// TIA Portal project "TrattamentiTermici" (V18)

(* hardware
DEVICE "S71500/ET200MP station_1"  S7-1500 station
   slot 0: "Telaio di montaggio_0"  Rack  6ES7 590-1***0-0AA0
   slot 1: "PLC_1"  CPU 1516-3 PN/DP  6ES7 516-3AN01-0AB0  V2.5
      slot 3: "Display CPU_1"  6ES7591-1BA00-0AA0
   slot 2: "DI 32x24VDC HF_1"  DI 32x24VDC HF  6ES7 521-1BL00-0AB0  V2.1
   slot 3: "DQ 32x24VDC/0.5A HF_1"  DQ 32x24VDC/0.5A HF  6ES7 522-1BL01-0AB0  V1.0
   slot 4: "AI 8xU/I/RTD/TC ST_1"  AI 8xU/I/RTD/TC ST  6ES7 531-7KF00-0AB0  V2.1
   slot 5: "AQ 4xU/I ST_1"  AQ 4xU/I ST  6ES7 532-5HD00-0AB0  V2.1
*)

// ===== PLC "PLC_1"  CPU 1516-3 PN/DP =====

VAR_GLOBAL   // PLC tag table "Tabella delle variabili standard"
   "AperturaCoperchio" AT %Q0.0 : Bool;
   "ChiusuraCoperchio" AT %Q0.1 : Bool;
   "DiscesaPunta" AT %Q0.2 : Bool;
   "AbbassaBraccio" AT %Q0.3 : Bool;
   "LedEmergenza" AT %Q0.4 : Bool;
   "MotoreIndietro" AT %Q0.5 : Bool;
   "MotoreAvanti" AT %Q0.6 : Bool;
   "SalitaPunta" AT %Q0.7 : Bool;
   "AlzaBraccio" AT %Q1.0 : Bool;
   "led11" AT %Q1.1 : Bool;
   "led12" AT %Q1.2 : Bool;
   "led13" AT %Q1.3 : Bool;
   "led14" AT %Q1.4 : Bool;
   "led15" AT %Q1.5 : Bool;
   "led16" AT %Q1.6 : Bool;
   "led17" AT %Q1.7 : Bool;
   "led20" AT %Q2.0 : Bool;
   "led21" AT %Q2.1 : Bool;
   "led22" AT %Q2.2 : Bool;
   "led23" AT %Q2.3 : Bool;
   "led24" AT %Q2.4 : Bool;
   "led25" AT %Q2.5 : Bool;
   "led26" AT %Q2.6 : Bool;
   "led27" AT %Q2.7 : Bool;
   "led30" AT %Q3.0 : Bool;
   "led31" AT %Q3.1 : Bool;
   "led32" AT %Q3.2 : Bool;
   "led33" AT %Q3.3 : Bool;
   "led34" AT %Q3.4 : Bool;
   "led35" AT %Q3.5 : Bool;
   "led36" AT %Q3.6 : Bool;
   "led37" AT %Q3.7 : Bool;
   "BraccioSu" AT %I0.2 : Bool;
   "BraccioGiu" AT %I0.3 : Bool;
   "FotocellulaSinistra" AT %I0.4 : Bool;
   "FotocellulaCentrale" AT %I0.5 : Bool;
   "FotocellulaDestra" AT %I0.6 : Bool;
   "PulsanteInizializzazione" AT %I0.7 : Bool;
   "PulsanteMarcia" AT %I1.0 : Bool;
   "PulsanteStop" AT %I1.1 : Bool;
   "PulsanteEmergenza" AT %I1.2 : Bool;
   "CoperchioAperto" AT %I2.1 : Bool;
END_VAR

DATA_BLOCK "DB_Comandi"   // DB1
{ S7_Optimized_Access := 'FALSE' }
VERSION : 0.1
   VAR
      bStop : Bool;
      bAuto : Bool;
      bMan : Bool;
      bReset : Bool;
      bEmergenza : Bool;
   END_VAR
BEGIN
END_DATA_BLOCK

DATA_BLOCK "DB_Stati"   // DB2
{ S7_Optimized_Access := 'FALSE' }
VERSION : 0.1
   VAR
      sAuto : Bool;
      sStop : Bool;
      sMan : Bool;
      sHome : Bool;
      sAttesastop : Bool;
      sEmergenza : Bool;
      bIni1 : Bool;
      bIni2 : Bool;
      bRip1 : Bool;
      bRip2 : Bool;
   END_VAR
BEGIN
END_DATA_BLOCK

DATA_BLOCK "DB_Tappe"   // DB3
{ S7_Optimized_Access := 'FALSE' }
VERSION : 0.1
   VAR
      tappeGemma : Int;
      tappeM1 : Int;
   END_VAR
BEGIN
END_DATA_BLOCK

DATA_BLOCK "DB_Variabili"   // DB4
{ S7_Optimized_Access := 'FALSE' }
VERSION : 0.1
   VAR
      timerResetPulsantiSTART : Bool;
      timerResetPulsantiDONE : Bool;
      timerResetPulsantiOUTPUT : Time;
      timerResetPulsantiDURATA : Time;
      BraccioSu : Bool;
      BraccioGiu : Bool;
      FotocellulaSinistra : Bool;
      FotocellulaCentrale : Bool;
      FotocellulaDestra : Bool;
      BtnInizio : Bool;
      BtnMarcia : Bool;
      BtnStop : Bool;
      BtnEmergenza : Bool;
      CoperchioAperto : Bool;
      AperturaCoperchio : Bool;
      ChiusuraCoperchio : Bool;
      DiscesaPunta : Bool;
      AbbassaBraccio : Bool;
      LedEmergenza : Bool;
      MotoreIndietro : Bool;
      MotoreAvanti : Bool;
      AlzaBraccio : Bool;
      SalitaPunta : Bool;
      nShake : Int;
      nPezzi : Int;
      giaAumentato : Bool;
   END_VAR
BEGIN
END_DATA_BLOCK

// folder: System blocks/Program resources

DATA_BLOCK "timerResetPulsanti"   // DB5
{ S7_Optimized_Access := 'TRUE' }
AUTHOR : Simatic
FAMILY : IEC
NAME : IEC_TMR
VERSION : 1.0
// stored: InstanceOfName IEC_TIMER
"IEC_TIMER"
BEGIN
END_DATA_BLOCK

// folder: (top level)

FUNCTION "FC_Gemma" : Void   // FC1, SCL
{ S7_Optimized_Access := 'TRUE' }
VERSION : 0.1
BEGIN
   CASE "DB_Tappe".tappeGemma OF
       0:  //Stato di riposo
           "DB_Stati".sStop := TRUE;
           IF "DB_Comandi".bAuto = TRUE THEN
               "DB_Tappe".tappeGemma := 1;//home
               "DB_Stati".sAuto := FALSE;
               "DB_Stati".sHome := TRUE;
               "DB_Stati".sMan := FALSE;
               "DB_Stati".sStop := FALSE;
               "DB_Stati".sEmergenza := FALSE;
           ELSE
               IF "DB_Comandi".bMan = TRUE THEN
                   "DB_Tappe".tappeGemma := 4;//home
                   "DB_Stati".sAuto := FALSE;
                   "DB_Stati".sHome := FALSE;
                   "DB_Stati".sMan := TRUE;
                   "DB_Stati".sStop := FALSE;
                   "DB_Stati".sEmergenza := FALSE;
               END_IF;
           END_IF;
          1: //Stato di home
              IF "DB_Stati".bIni1 = TRUE AND "DB_Stati".bIni2 = TRUE THEN
                  "DB_Tappe".tappeGemma := 2;//automatico
                  "DB_Stati".sAttesastop := TRUE;
                  "DB_Stati".sAuto := TRUE;
                  "DB_Stati".sHome := FALSE;
                  "DB_Stati".sMan := FALSE;
                  "DB_Stati".sStop := FALSE;
                  "DB_Stati".sEmergenza := FALSE;
              END_IF;
          2: //Stato di automatico
              IF "DB_Comandi".bStop = TRUE THEN
                  "DB_Tappe".tappeGemma := 3;//attesa stop
                  "DB_Stati".sAttesastop := TRUE;
                  "DB_Stati".sAuto := FALSE;
                  "DB_Stati".sHome := FALSE;
                  "DB_Stati".sMan := FALSE;
                  "DB_Stati".sStop := FALSE;
                  "DB_Stati".sEmergenza := FALSE;
              END_IF;
          3: //Stato di attesa stop
              IF "DB_Stati".bRip1 = TRUE AND "DB_Stati".bRip2 = TRUE THEN
                  "DB_Tappe".tappeGemma := 0;//stop
                  "DB_Stati".sAttesastop := TRUE;
                  "DB_Stati".sAuto := FALSE;
                  "DB_Stati".sHome := FALSE;
                  "DB_Stati".sMan := FALSE;
                  "DB_Stati".sStop := TRUE;
                  "DB_Stati".sEmergenza := FALSE;
              END_IF;
          4: //Stato di manuale
              IF "DB_Comandi".bStop = TRUE = TRUE THEN
                  "DB_Tappe".tappeGemma := 0;//stop
                  "DB_Stati".sAuto := FALSE;
                  "DB_Stati".sHome := FALSE;
                  "DB_Stati".sMan := FALSE;
                  "DB_Stati".sStop := TRUE;
                  "DB_Stati".sEmergenza := FALSE;
              END_IF;
          5: //Stato di emergenza
              IF "DB_Comandi".bEmergenza = TRUE AND "DB_Stati".sEmergenza = TRUE THEN
                  "DB_Tappe".tappeGemma := 0;//stop
                  "DB_Stati".sAuto := FALSE;
                  "DB_Stati".sHome := FALSE;
                  "DB_Stati".sMan := FALSE;
                  "DB_Stati".sStop := TRUE;
                  "DB_Stati".sEmergenza := FALSE;
              END_IF;
      END_CASE;
   //gestione emergenza

      IF "DB_Comandi".bEmergenza = FALSE THEN
          "DB_Tappe".tappeGemma := 5;//emergenza
      "DB_Stati".sAttesastop := FALSE;
      "DB_Stati".sAuto := FALSE;
      "DB_Stati".sHome := FALSE;
      "DB_Stati".sMan := FALSE;
      "DB_Stati".sStop := FALSE;
      "DB_Stati".sEmergenza := TRUE;
   END_IF;
END_FUNCTION

FUNCTION "FC_Grafcet" : Void   // FC2, SCL
{ S7_Optimized_Access := 'TRUE' }
VERSION : 0.1
BEGIN
   //Imposto bRini e bRip a TRUE. Andranno poi gestiti in base alle condizioni dell'impianto
   "DB_Stati".bIni1 := TRUE;
   "DB_Stati".bIni2 := TRUE;
   "DB_Stati".bRip1 := TRUE;
   "DB_Stati".bRip2 := TRUE;
   //
   //gestico il RESET
   //

   IF "DB_Tappe".tappeM1 = 0 THEN
       IF "DB_Stati".sAuto AND "DB_Stati".bIni1 AND "DB_Stati".sAttesastop THEN
           "DB_Tappe".tappeM1 := 1;
       END_IF;

       "DB_Variabili".nPezzi := 0;
       "DB_Variabili".timerResetPulsantiDURATA := T#400ms;
   END_IF;

   IF "DB_Tappe".tappeM1 = 1 THEN
       "DB_Variabili".AlzaBraccio := TRUE;

       IF "DB_Variabili".BraccioSu  THEN
           "DB_Variabili".AlzaBraccio := FALSE;
           "DB_Variabili".MotoreAvanti := TRUE;
       END_IF;

       IF "DB_Variabili".FotocellulaCentrale=TRUE THEN
           "DB_Variabili".MotoreAvanti := FALSE;
           "DB_Tappe".tappeM1 := 2;
       END_IF;
   END_IF;

   IF "DB_Tappe".tappeM1 = 2 THEN
       "DB_Variabili".AbbassaBraccio := TRUE;
       "DB_Variabili".nShake := 0;

       IF "DB_Variabili".BraccioGiu THEN
           "DB_Variabili".AbbassaBraccio := FALSE;
           "DB_Tappe".tappeM1 := 3;
           "DB_Variabili".nShake := 0;
       END_IF;
   END_IF;


   IF "DB_Tappe".tappeM1 = 3 THEN
       "DB_Variabili".DiscesaPunta := TRUE;
       "DB_Variabili".timerResetPulsantiDURATA := T#400ms;
       "DB_Variabili".timerResetPulsantiSTART := TRUE;

       IF "DB_Variabili".timerResetPulsantiDONE THEN
           "DB_Variabili".timerResetPulsantiSTART := FALSE;
           "DB_Variabili".timerResetPulsantiDONE := FALSE;
           "DB_Variabili".giaAumentato := FALSE;
           "DB_Variabili".DiscesaPunta := FALSE;
           "DB_Tappe".tappeM1 := 4;
       END_IF;
   END_IF;

   IF "DB_Tappe".tappeM1 = 4 THEN
       "DB_Variabili".SalitaPunta := TRUE;
       "DB_Variabili".timerResetPulsantiSTART := TRUE;
       "DB_Variabili".timerResetPulsantiDURATA := T#400ms;

       IF "DB_Variabili".timerResetPulsantiDONE THEN
           IF "DB_Variabili".giaAumentato=FALSE THEN
               "DB_Variabili".nShake += 1;
               "DB_Variabili".giaAumentato := TRUE;
               "DB_Variabili".SalitaPunta := FALSE;
           END_IF;
           IF "DB_Variabili".nShake = 6 THEN
               "DB_Variabili".AlzaBraccio := TRUE;
               IF "DB_Variabili".BraccioSu THEN
                   "DB_Variabili".AlzaBraccio := FALSE;
                   "DB_Variabili".timerResetPulsantiSTART := FALSE;
                   "DB_Variabili".timerResetPulsantiDONE := FALSE;
                   "DB_Tappe".tappeM1 := 5;
               END_IF;
           ELSE
               "DB_Tappe".tappeM1 := 3;
           END_IF;
       END_IF;
   END_IF;

   IF "DB_Tappe".tappeM1 = 5 THEN
       "DB_Variabili".AperturaCoperchio := TRUE;
       "DB_Variabili".MotoreAvanti := TRUE;

       IF "DB_Variabili".FotocellulaDestra = TRUE THEN
           "DB_Variabili".AperturaCoperchio := FALSE;
           "DB_Variabili".MotoreAvanti := FALSE;
           "DB_Tappe".tappeM1 := 6;
       END_IF;
   END_IF;

   IF "DB_Tappe".tappeM1 = 6 THEN
       "DB_Variabili".AbbassaBraccio := TRUE;

       IF "DB_Variabili".BraccioGiu THEN
           "DB_Variabili".AbbassaBraccio := FALSE;
           "DB_Variabili".DiscesaPunta := TRUE;
           "DB_Variabili".timerResetPulsantiSTART := TRUE;
           "DB_Variabili".timerResetPulsantiDURATA := T#3000ms;
       END_IF;

       IF "DB_Variabili".timerResetPulsantiDONE THEN
           "DB_Variabili".DiscesaPunta := FALSE;
           "DB_Variabili".timerResetPulsantiSTART := FALSE;
           "DB_Variabili".timerResetPulsantiDONE := FALSE;
           "DB_Tappe".tappeM1 := 7;
       END_IF;
   END_IF;

   IF "DB_Tappe".tappeM1 = 7 THEN
       "DB_Variabili".SalitaPunta := TRUE;
       "DB_Variabili".AlzaBraccio := TRUE;

       IF "DB_Variabili".BraccioSu THEN
           "DB_Variabili".SalitaPunta := FALSE;
           "DB_Variabili".AlzaBraccio := FALSE;
           "DB_Tappe".tappeM1 := 8;
           "DB_Variabili".nPezzi+=1;
       END_IF;
       ;
   END_IF;

   IF "DB_Tappe".tappeM1 = 8 THEN
       "DB_Variabili".MotoreIndietro := TRUE;

       IF "DB_Variabili".FotocellulaCentrale THEN
           "DB_Variabili".MotoreIndietro := FALSE;
           "DB_Tappe".tappeM1 := 9;
       END_IF;
       ;
   END_IF;

   IF "DB_Tappe".tappeM1 = 9 THEN
       "DB_Variabili".MotoreIndietro := TRUE;
       "DB_Variabili".ChiusuraCoperchio := TRUE;

       IF "DB_Variabili".FotocellulaSinistra THEN
           "DB_Variabili".MotoreIndietro := FALSE;
           "DB_Variabili".timerResetPulsantiSTART := TRUE;
           "DB_Variabili".timerResetPulsantiDONE := FALSE;
           "DB_Variabili".timerResetPulsantiDURATA := T#5000ms;
       END_IF;

       IF "DB_Variabili".timerResetPulsantiDONE THEN
           "DB_Variabili".timerResetPulsantiSTART := FALSE;
           "DB_Variabili".timerResetPulsantiDONE := FALSE;
           "DB_Tappe".tappeM1 := 0;
           "DB_Variabili".ChiusuraCoperchio := FALSE;
       END_IF;
   END_IF;
END_FUNCTION

FUNCTION "FC_ResetPulsanti" : Void   // FC3, SCL
{ S7_Optimized_Access := 'TRUE' }
VERSION : 0.1
BEGIN
   IF "DB_Comandi".bAuto = TRUE OR
       "DB_Comandi".bMan = TRUE OR
       "DB_Comandi".bReset = TRUE OR
       "DB_Comandi".bStop = TRUE THEN
       //
       "DB_Variabili".timerResetPulsantiSTART := TRUE;
   END_IF;
   IF "DB_Variabili".timerResetPulsantiDONE = TRUE THEN
       "DB_Variabili".timerResetPulsantiSTART := FALSE;
       "DB_Variabili".timerResetPulsantiDONE := FALSE;
       "DB_Comandi".bAuto := FALSE;
       "DB_Comandi".bMan := FALSE;
       "DB_Comandi".bReset := FALSE;
       "DB_Comandi".bStop := FALSE;
   END_IF;
END_FUNCTION

FUNCTION "FC_Timer" : Void   // FC4, SCL
{ S7_Optimized_Access := 'TRUE' }
VERSION : 0.1
BEGIN
   "DB_Variabili".timerResetPulsantiDURATA := T#400ms;
   "timerResetPulsanti".TON(IN:="DB_Variabili".timerResetPulsantiSTART,
                            PT:="DB_Variabili".timerResetPulsantiDURATA,
                            Q=>"DB_Variabili".timerResetPulsantiDONE,
                            ET=>"DB_Variabili".timerResetPulsantiOUTPUT);
END_FUNCTION

FUNCTION "FC_Uscite" : Void   // FC5, SCL
{ S7_Optimized_Access := 'TRUE' }
VERSION : 0.1
BEGIN
   //prima di scrivere fisicamente le uscite
   //devo controllare che tutte le condizioni
   //siano rispettate
   //emergenza, protezioni, fotocellule ecc.
   "AperturaCoperchio" := "DB_Variabili".ChiusuraCoperchio;
   "ChiusuraCoperchio" := "DB_Variabili".AperturaCoperchio;
   "DiscesaPunta" := "DB_Variabili".AbbassaBraccio;
   "AbbassaBraccio" := "DB_Variabili".DiscesaPunta;
   "LedEmergenza" := "DB_Variabili".LedEmergenza;
   "MotoreIndietro" := "DB_Variabili".MotoreIndietro;
   "MotoreAvanti" := "DB_Variabili".MotoreAvanti;
   "AlzaBraccio" := "DB_Variabili".AlzaBraccio;
   "SalitaPunta" := "DB_Variabili".SalitaPunta;

   // Uscite
   "DB_Variabili".BraccioSu := "BraccioSu";
   "DB_Variabili".BraccioGiu := "BraccioGiu";
   "DB_Variabili".FotocellulaSinistra := "FotocellulaSinistra";
   "DB_Variabili".FotocellulaCentrale := "FotocellulaCentrale";
   "DB_Variabili".FotocellulaDestra := "FotocellulaDestra";
   "DB_Variabili".BtnInizio := "PulsanteMarcia";
   "DB_Variabili".BtnStop := "PulsanteStop";
   "DB_Variabili".BtnEmergenza := "PulsanteEmergenza";
   "DB_Variabili".CoperchioAperto :="CoperchioAperto";
END_FUNCTION

ORGANIZATION_BLOCK "Main"   // OB1, LAD, ProgramCycle
TITLE = "Main Program Sweep (Cycle)"
{ S7_Optimized_Access := 'TRUE' }
VERSION : 0.1
   VAR_INPUT
      Initial_Call : Bool;   // Initial call of this OB
      Remanence : Bool;   // =True, if remanent data are available
   END_VAR
   VAR_TEMP   // added for the SCL form of the ladder/FBD networks
      _w1 : Bool;
      _w2 : Bool;
      _w3 : Bool;
      _w4 : Bool;
   END_VAR
BEGIN

REGION Network 1
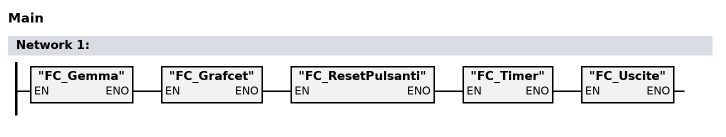
   RUNG wire#powerrail
      "FC_Gemma"()
      "FC_Grafcet"()
      "FC_ResetPulsanti"()
      "FC_Timer"()
      "FC_Uscite"()
   END_RUNG
   // the same network as SCL:
   "FC_Gemma"(ENO => #_w1);
   "FC_Grafcet"(EN := #_w1, ENO => #_w2);
   "FC_ResetPulsanti"(EN := #_w2, ENO => #_w3);
   "FC_Timer"(EN := #_w3, ENO => #_w4);
   IF #_w4 THEN "FC_Uscite"(); END_IF;
END_REGION
END_ORGANIZATION_BLOCK